// TIA Portal V17 export
// export: Created 2025-03-12T15:37:02.7798916Z, ExportSetting WithDefaults, DisplayName Totally Integrated Automation Portal, DisplayVersion V17 Update 8, DisplayName TIA Portal Openness, DisplayVersion V17 Update 8, DisplayName TIA Portal Version Control Interface, DisplayVersion V17, DisplayName SINAMICS Startdrive Advanced, DisplayVersion V17 SP2, DisplayName SINAMICS Startdrive G110M, G120, G120C, G120D, G120P, G115D, DisplayVersion V17 SP2, DisplayName SINAMICS Startdrive G130, G150, S120, S150, SINAMICS MV, S210, DisplayVersion V17 SP2, DisplayName STEP 7 Professional, DisplayVersion V17 Update 8, DisplayName SINUMERIK ONE STEP 7 Toolbox, DisplayVersion V17 Update 12, DisplayName SINUMERIK 840D sl STEP 7 Toolbox, DisplayVersion V17 Update 12, DisplayName STEP 7 Safety, DisplayVersion V17 Update 6, DisplayName WinCC Advanced, DisplayVersion V17 Update 8
TYPE "OPEN_CLOSE_HATCH_CLADDING"
// stored: IsFailsafeCompliant false
   STRUCT
      GENERAL_CONDITIONS : Bool;   // GENERAL CONDITIONS
      CLOSE_CONDITIONS : Bool;   // ADVANCE CONDITIONS / CLOSE CONDITIONS
      OPEN_CONDITIONS : Bool;   // RETURN CONDITIONS / OPEN CONDITIONS
      GENERAL_CONDITIONS_HELP : Bool;   // GENERAL CONDITIONS HELP
      CLOSE_CONDITIONS_HELP : Bool;   // CLOSE CONDITIONS HELP
      OPEN_CONDITIONS_HELP : Bool;   // OPEN CONDITIONS HELP
      CLOSE_HMI_REQUEST : Bool;   // ADVANCE HMI REQUEST / CLOSE MANUAL HMI REQUEST
      OPEN_HMI_REQUEST : Bool;   // RETURN HMI REQUEST / OPEN MANUAL HMI REQUEST
      CLOSE_MANUAL_REQUEST : Bool;   // ADVANCE MANUAL REQUEST / CLOSE MANUAL REQUEST
      OPEN_MANUAL_REQUEST : Bool;   // RETURN MANUAL REQUEST / OPEN MANUAL REQUEST
      CLOSE_AUTO_REQUEST : Bool;   // ADVANCE AUTO REQUEST / CLOSE AUTO REQUEST
      OPEN_AUTO_REQUEST : Bool;   // RETURN AUTO REQUEST / OPEN AUTO REQUEST
      CLOSE_GLOBAL_REQUEST : Bool;   // ADVANCE GLOBAL REQUEST / CLOSE GLOBAL REQUEST
      OPEN_GLOBAL_REQUEST : Bool;   // RETURN GLOBAL REQUEST / OPEN GLOBAL REQUEST
      CLOSE_COMMAND : Bool;   // ADVANCE COMMAND / CLOSE COMMAND
      OPEN_COMMAND : Bool;   // RETURN COMMAND / OPEN COMMAND
      FULL_CLOSED : Bool;   // ADVANCED FEEDBACK / CLOSED AND COMMANDED
      FULL_OPENED : Bool;   // RETURNED FEEDBACK / OPENED AND COMMANDED
      SIMULTANEITY_ALARM : Bool;   // SIMULTANEITY FAULT / SIMULTANEITY ALARM
      TIME_EXCEEDED_ALARM : Bool;   // TIME EXCEEDED / TIME EXCEEDED ALARM
      ANY_ACTIVE_ALARM : Bool;   // FAULT / ANY ACTIVE ALARM
      IS_SEOC_ALARMS : Bool;   // INMEDIATE STOP AND STOP END OF CYCLE ALARMS
      PULSE_1 : Bool;   // PULSE 1
      PULSE_2 : Bool;   // PULSE 2
      PULSE_3 : Bool;   // PULSE 3
   END_STRUCT;
END_TYPE
